// TIA Portal V20 export
TYPE "typeCmControlNodeSoftCam"
// stored: Namespace Unit1.Em4
   STRUCT
      sideTapeFixStageAxisX : "Unit1.Em4.typeCmControlNodeSoftCamsideTapeFixStageAxisX";
      sideTapeFixStageAxisC : "Unit1.Em4.typeCmControlNodeSoftCamsideTapeFixStageAxisC";
      sideTapeAttachmentAxisX : "Unit1.Em4.typeCmControlNodeSoftCamsideTapeAttachmentAxisX";
      sideTapeAttachmentAxisY : "Unit1.Em4.typeCmControlNodeSoftCamsideTapeAttachmentAxisY";
   END_STRUCT;
END_TYPE
